RoboDK station: Engraving my Full Name.rdk

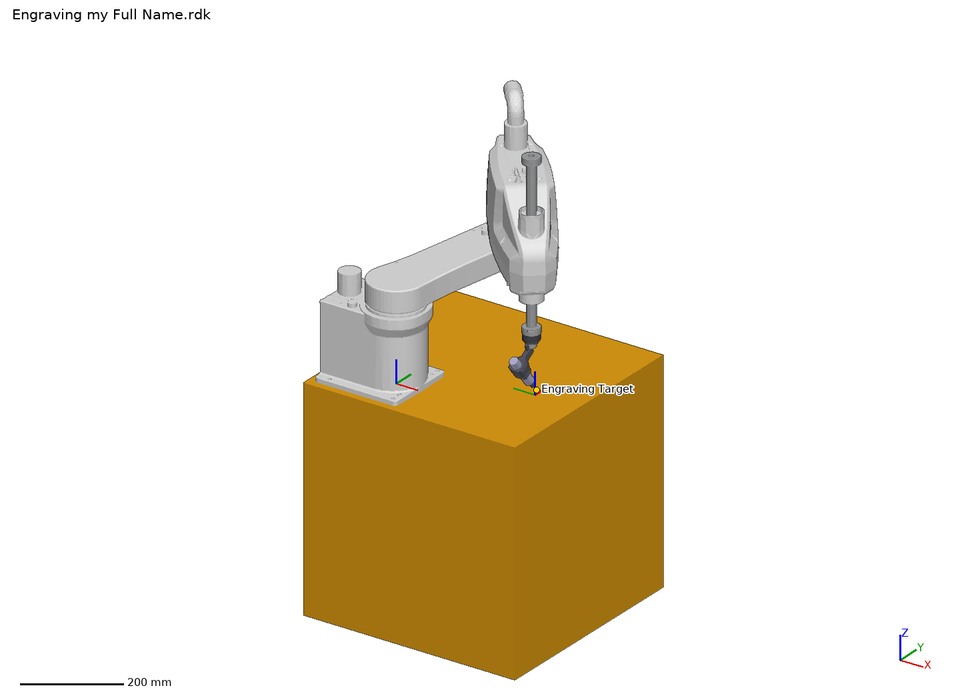
[picture v0: the station drawn from its stored meshes, robots at their saved joint values, targets as dots, program paths as lines]
Station Engraving my Full Name (saved by RoboDK 5.3.0). Poses are relative to the parent item; angles as X-Y-Z fixed-axis rotations.
  - frame Mitsubishi RH-6CH60 Base at (0, 0, 0) mm
    - robot Mitsubishi RH-6CH60: 4 axes, payload 6 kg, reach 600 mm, repeatability 0.025 mm, weight 17 kg
        modified DH rows (alpha deg, a mm, theta deg, d mm): 0, 0, 0, 0; 0, 325, 0, 0; 0, 275, 0, -50 linear; 180, 0, 0, 0
        joint limits [-132, -150, 0, -360] to [132, 150, 200, 360]; home [0, 0, 200, 0]; saved at [79.785, -128.414, 151.508, 133.405]
      - tool Spindle, TCP at (15.83, 0, -100.51) mm, size 78.7 x 36 x 130 mm
  - object Cube 500mm at (-150, -100, 0) mm, size 500 x 500 x 500 mm, geometry from Cube-500mm.sld
    - object A4-Paper at (500, 500, 1) mm, rotated rx -90 ry 0 rz 180 deg, geometry from A4-Paper.STL
      - item type 7 A4-Paper-0
      - item type 7 A4-Paper-1
  - frame Starting Frame at (250, 110, 1) mm, rotated rx 0 ry 0 rz 90 deg
    - target Engraving Target (Cartesian target) at (19.24, 9.17, 0) mm, rotated rx 0 ry 0 rz -5.22 deg; joints [-55.246, -12.237, 126.374, 62.259] of Mitsubishi RH-6CH60
  - Python program Engraving Program (listed below)

--- Python program Engraving Program ---
from robolink import *    # RoboDK API
from robodk import *      # Robot toolbox

data = LoadList("my name.csv") #Reading the points from the CSV file

#Defining the Robot
RDK = Robolink()
robot = RDK.Item('',ITEM_TYPE_ROBOT)

#Defining the Engraving Frame and the Starting Point and Moving te robot to the starting position
frame = RDK.Item('Starting Frame')
target = RDK.Item('Engraving Target')
TarPose = target.Pose()
robot.setPoseFrame(frame)

#Asking the user to Check the tracing style to Line
RDK.ShowMessage('''PLease change the tracing style to Line
                    Go to: Tools -> Trace -> Style -> Line''')

#Moving the robot through the obtained points from the csv
for i in range(len(data)):
    TarPose.setPos(data[i])
    target.setPose(TarPose)

    #Activating the Trace if the engraving on the XY plan and Deactiviting the Trace otherwise
    if (data[i][2] == 0 )and (data[i-1][2] ==0):
        RDK.Command("Trace", "On")
        robot.MoveL(target)
    else:
        RDK.Command("Trace", "Off")
        robot.MoveJ(target)
    if i == 0:
        RDK.Command("Trace", "Reset")


#Notifying the user that the engraving is done
RDK.ShowMessage("Done Engraving")
